(* IEC 61131-3 sources: lc3-arduino-ethernet/src, 3 files *)

(* ---- ControllinoMaxiAutomationHwInfo.iecst ---- *)
/*
 * Number of LEDs for Controllino MAXI Automation platform
 */
FUNCTION GetNumberOfLEDs: USINT
	GetNumberOfLEDs := 18;
END_FUNCTION

FUNCTION GetNumberOfInputs: USINT
	GetNumberOfInputs := 4;
END_FUNCTION

FUNCTION ControllinoMapDigitalInputIdxToPin : USINT
	VAR_INPUT
		index : USINT;
	END_VAR
	CASE index OF
		0 : ControllinoMapDigitalInputIdxToPin := ControllinoMaxiAutomationDigital#I0;
		1 : ControllinoMapDigitalInputIdxToPin := ControllinoMaxiAutomationDigital#I1;
		2 : ControllinoMapDigitalInputIdxToPin := ControllinoMaxiAutomationDigital#I2;
		3 : ControllinoMapDigitalInputIdxToPin := ControllinoMaxiAutomationDigital#I3;
	ELSE
		ENO := FALSE;
	END_CASE;
END_FUNCTION

FUNCTION ControllinoMapDigitalOutputIdxToPin : USINT
	VAR_INPUT
		index : USINT;
	END_VAR
	CASE index OF
		 0 : ControllinoMapDigitalOutputIdxToPin := ControllinoMaxiAutomationDigital#D0;
		 1 : ControllinoMapDigitalOutputIdxToPin := ControllinoMaxiAutomationDigital#D1;
		 2 : ControllinoMapDigitalOutputIdxToPin := ControllinoMaxiAutomationDigital#D2;
		 3 : ControllinoMapDigitalOutputIdxToPin := ControllinoMaxiAutomationDigital#D3;
		 4 : ControllinoMapDigitalOutputIdxToPin := ControllinoMaxiAutomationDigital#D4;
		 5 : ControllinoMapDigitalOutputIdxToPin := ControllinoMaxiAutomationDigital#D5;
		 6 : ControllinoMapDigitalOutputIdxToPin := ControllinoMaxiAutomationDigital#D6;
		 7 : ControllinoMapDigitalOutputIdxToPin := ControllinoMaxiAutomationDigital#D7;
		 8 : ControllinoMapDigitalOutputIdxToPin := ControllinoMaxiAutomationDigital#R0;
		 9 : ControllinoMapDigitalOutputIdxToPin := ControllinoMaxiAutomationDigital#R1;
		10 : ControllinoMapDigitalOutputIdxToPin := ControllinoMaxiAutomationDigital#R2;
		11 : ControllinoMapDigitalOutputIdxToPin := ControllinoMaxiAutomationDigital#R3;
		12 : ControllinoMapDigitalOutputIdxToPin := ControllinoMaxiAutomationDigital#R4;
		13 : ControllinoMapDigitalOutputIdxToPin := ControllinoMaxiAutomationDigital#R5;
		14 : ControllinoMapDigitalOutputIdxToPin := ControllinoMaxiAutomationDigital#R6;
		15 : ControllinoMapDigitalOutputIdxToPin := ControllinoMaxiAutomationDigital#R7;
		16 : ControllinoMapDigitalOutputIdxToPin := ControllinoMaxiAutomationDigital#R8;
		17 : ControllinoMapDigitalOutputIdxToPin := ControllinoMaxiAutomationDigital#R9;
	ELSE
		ENO := FALSE;
	END_CASE;
END_FUNCTION

(* ---- HandleEthernet.iecfbd ---- *)
FUNCTION_BLOCK HandleEthernet
  VAR
    mac : ADDR_MAC := [16#DE, 16#AD, 16#BE, 16#EF, 16#FE, 16#ED];
    ip : ADDR_IP := [192, 168, 99, 123];
    tcpPort : ADDR_PORT := 80;
    init : BOOL := TRUE;
  END_VAR

  (*

    // Network 1:
    EthernetBegin(mac := mac, ip := ip, tcp_port := tcpPort, enable := init, success => @C(1).success);
    NOT(IN := @C(1).success, NOT => init);

    // Network 2:
    NOT(IN := init, NOT => @C(7).NOT);
    EthernetServer(enable := @C(7).NOT);

  *)

  @C(1) : @F(EthernetBegin), @R(450.0, 110.0, 270.0, 78.0), @I(@N(mac), @L(9.5)), @I(@N(ip), @L(29.5)), @I(@N(tcp_port), @L(49.5)), @I(@N(enable), @L(69.5)), @O(@N(success), @R(9.5));
  @C(2) : @F(EthernetServer), @R(450.0, 230.0, 120.0, 78.0), @I(@N(enable), @L(9.5)), @O(@N(success), @R(9.5));
  @VF(4) : @E(mac), @R(170.0, 110.0, 140.0, 19.0);
  @VF(8) : @E(ip), @R(170.0, 130.0, 140.0, 19.0);
  @VF(9) : @E(tcpPort), @R(170.0, 150.0, 140.0, 19.0);
  @VF(3) : @E(init), @R(170.0, 170.0, 140.0, 19.0);
  @VF(6) : @E(init), @R(880.0, 110.0, 140.0, 19.0);
  @VF(13) : @E(init), @R(170.0, 230.0, 140.0, 19.0);
  @C(7) : @F(NOT), @R(350.0, 230.0, 60.0, 18.5), BOOL, @I(@N(IN), @L(9.5)), @O(@N(NOT), @R(9.5));
  @C(16) : @F(NOT), @R(780.0, 110.0, 60.0, 18.5), BOOL, @I(@N(IN), @L(9.5)), @O(@N(NOT), @R(9.5));

  @G(10) :
     @L(@VF(4).o, @C(1).mac)
    ;
  @G(11) :
     @L(@VF(8).o, @C(1).ip)
    ;
  @G(12) :
     @L(@VF(9).o, @C(1).tcp_port)
    ;
  @G(5) :
     @L(@VF(3).o, @C(1).enable)
    ;
  @G(14) :
     @L(@C(7).NOT, @C(2).enable)
    ;
  @G(15) :
     @L(@VF(13).o, @C(7).IN)
    ;
  @G(17) :
     @L(@C(1).success, @C(16).IN)
    ;
  @G(18) :
     @L(@C(16).NOT, @VF(6).i)
    ;
END_FUNCTION_BLOCK

(* ---- program.iecst ---- *)
/*
 * This is the main program for the Controllino moving light example. <br/>
 * The following steps are performed:                                 <br/>
 * - initialize the Controllino system (called only once)             <br/>
 * - read inputs                                                      <br/>
 * - execute program logic                                            <br/>
 * - write outputs                                                    <br/>
 */
PROGRAM ControllinoMovingLight
	VAR_GLOBAL
		switchInvert : BOOL;
		outLedPattern : LWORD;
	END_VAR

	VAR
		isInitialized : BOOL;
		movingLight : MovingLight;
		ethernet : HandleEthernet;
	END_VAR

	IF NOT isInitialized THEN
		ControllinoInitialize(ENO => isInitialized);
	END_IF;

	MapInputsToVariables();
	movingLight(numberOfLEDs := GetNumberOfLEDs());
	MapVariablesToOutputs();

	ethernet();

END_PROGRAM
